// TIA Portal V20 export
TYPE "type_emRelations_em3_sequence"
// stored: Access Published, Namespace Unit1
   STRUCT
      topTapeLoading : Struct
         jobs : "LAF_typeJobs";
         sequence : "LAF_typeSequence";
         selectJobStatus { S7_SetPoint := 'True'} : Array[0..10] of "LAF_typeJobStatus";
         "step" : "LER_typeStep";
         jobInterface : Struct
            chargeJob2 : "LER_typeJobInterface";
         END_STRUCT;
         homeCheck : Struct
            TapeLoadReq { ExternalWritable := 'False'} : Bool;
            TapeLoaded { ExternalWritable := 'False'} : Bool;
         END_STRUCT;
      END_STRUCT;
      topTapeAttachment : Struct
         jobs : "LAF_typeJobs";
         sequence : "LAF_typeSequence";
         selectJobStatus { S7_SetPoint := 'True'} : Array[0..10] of "LAF_typeJobStatus";
         "step" : "LER_typeStep";
         jobInterface : Struct
            tapeGetJob2 : "LER_typeJobInterface";
            tape1PutJob3 : "LER_typeJobInterface";
            tape2PutJob4 : "LER_typeJobInterface";
            tapeIdleJob5 { S7_SetPoint := 'True'} : "LER_typeJobInterface";
         END_STRUCT;
         homeCheck : Struct
            tapeGetReq { ExternalWritable := 'False'} : Bool;
            tapeGet { ExternalWritable := 'False'} : Bool;
         END_STRUCT;
      END_STRUCT;
      topTapeFixStage : Struct
         jobs : "LAF_typeJobs";
         sequence : "LAF_typeSequence";
         selectJobStatus { S7_SetPoint := 'True'} : Array[0..10] of "LAF_typeJobStatus";
         "step" : "LER_typeStep";
         jobInterface : Struct
            loadJob2 : "LER_typeJobInterface";
            taping1Job3 : "LER_typeJobInterface";
            taping2Job4 : "LER_typeJobInterface";
            unloadJob5 : "LER_typeJobInterface";
         END_STRUCT;
         homeCheck : Struct
            partNoDetect { ExternalWritable := 'False'} : Bool;
            partDetect { ExternalWritable := 'False'} : Bool;
         END_STRUCT;
      END_STRUCT;
   END_STRUCT;
   // // topTapeLoading."step".action1[101] : Step[101] : JOB[1] Condition
   // // topTapeLoading."step".action1[110] : Step[110] : Top Tape Loading Backward
   // // topTapeLoading."step".action1[120] : Step[120] : Top Tape Loading Clamp Open
   // // topTapeLoading."step".action1[130] : Step[130] : Top Tape Cutter Up
   // // topTapeLoading."step".action1[140] : Step[140] : Top Tape Cutter Clamp Down
   // // topTapeLoading."step".action1[150] : Step[150] : Top Tape Tension Backward
   // // topTapeLoading."step".action1[190] : Step[190] : JOB[1] Step End
   // // topTapeLoading."step".action1[201] : Step[201] : JOB[2] Condition
   // // topTapeLoading."step".action1[210] : Step[210] : Top Tape Loading Forward & Tension Backward
   // // topTapeLoading."step".action1[220] : Step[220] : Top Tape Clamp Close
   // // topTapeLoading."step".action1[230] : Step[230] : Top Tape Cutter Clamp Up
   // // topTapeLoading."step".action1[240] : Step[240] : Top Tape Loading Backward & Tension Forward
   // // topTapeLoading."step".action1[250] : Step[250] : Top Tape Cutter Clamp Down
   // // topTapeLoading."step".action1[260] : Step[260] : Top Tape Tension Backward
   // // topTapeLoading."step".action1[290] : Step[290] : JOB[2] Step End
   // // topTapeLoading."step".transition1[101] : Step[101] : JOB[1] Condition
   // // topTapeLoading."step".transition1[110] : Step[110] : Top Tape Loading Backward
   // // topTapeLoading."step".transition1[120] : Step[120] : Top Tape Loading Clamp Open
   // // topTapeLoading."step".transition1[130] : Step[130] : Top Tape Cutter Up
   // // topTapeLoading."step".transition1[140] : Step[140] : Top Tape Cutter Clamp Down
   // // topTapeLoading."step".transition1[150] : Step[150] : Top Tape Tension Backward
   // // topTapeLoading."step".transition1[190] : Step[190] : JOB[1] Step End
   // // topTapeLoading."step".transition1[201] : Step[201] : JOB[2] Condition
   // // topTapeLoading."step".transition1[210] : Step[210] : Top Tape Loading Forward & Tension Backward
   // // topTapeLoading."step".transition1[220] : Step[220] : Top Tape Clamp Close
   // // topTapeLoading."step".transition1[230] : Step[230] : Top Tape Cutter Clamp Up
   // // topTapeLoading."step".transition1[240] : Step[240] : Top Tape Loading Backward & Tension Forward
   // // topTapeLoading."step".transition1[250] : Step[250] : Top Tape Cutter Clamp Down
   // // topTapeLoading."step".transition1[260] : Step[260] : Top Tape Tension Backward
   // // topTapeLoading."step".transition1[290] : Step[290] : JOB[2] Step End
   // // topTapeAttachment."step".action1[101] : Step[101] : JOB[1] Condition
   // // topTapeAttachment."step".action1[110] : Step[110] : Attachment Up
   // // topTapeAttachment."step".action1[120] : Step[120] : Top Tape X-Axis Remains Attach Pos
   // // topTapeAttachment."step".action1[130] : Step[130] : Top Tape Attachment Down
   // // topTapeAttachment."step".action1[140] : Step[140] : Top Tape Attachment Vaccum Off
   // // topTapeAttachment."step".action1[150] : Step[150] : Top Tape Attachment Up
   // // topTapeAttachment."step".action1[180] : Step[180] : Top Tape X-Axis Wait Pos
   // // topTapeAttachment."step".action1[190] : Step[190] : JOB[1] Step End
   // // topTapeAttachment."step".action1[201] : Step[201] : JOB[2] Condition
   // // topTapeAttachment."step".action1[210] : Step[210] : Top Tape X-Axis Wait Pos
   // // topTapeAttachment."step".action1[220] : Step[220] : Top Tape Attachment Down
   // // topTapeAttachment."step".action1[230] : Step[230] : Top Tape Attachment Vaccum On
   // // topTapeAttachment."step".action1[240] : Step[240] : Top Tape Cutter Down
   // // topTapeAttachment."step".action1[241] : Step[241] : Top Tape Cutter Up
   // // topTapeAttachment."step".action1[242] : Step[242] : Top Tape Clamp Open
   // // topTapeAttachment."step".action1[250] : Step[250] : Top Tape Attachment Up
   // // topTapeAttachment."step".action1[290] : Step[290] : JOB[2] Step End
   // // topTapeAttachment."step".action1[301] : Step[301] : JOB[3] Condition
   // // topTapeAttachment."step".action1[310] : Step[310] : Top Tape X-Axis Tape-1 Pos
   // // topTapeAttachment."step".action1[320] : Step[320] : Top Tape Attachment Down
   // // topTapeAttachment."step".action1[330] : Step[330] : Top Tape Attachment Vaccum Off
   // // topTapeAttachment."step".action1[370] : Step[370] : Top Tape Attachment Up
   // // topTapeAttachment."step".action1[380] : Step[380] : Top Tape X-Axis Wait Pos
   // // topTapeAttachment."step".action1[390] : Step[390] : JOB[3] Step End
   // // topTapeAttachment."step".action1[401] : Step[401] : JOB[4] Condition
   // // topTapeAttachment."step".action1[410] : Step[410] : Top Tape X-Axis Tape-2 Pos
   // // topTapeAttachment."step".action1[420] : Step[420] : Top Tape Attachment Down
   // // topTapeAttachment."step".action1[430] : Step[430] : Top Tape Attachment Vaccum Off
   // // topTapeAttachment."step".action1[470] : Step[470] : Top Tape Attachment Up
   // // topTapeAttachment."step".action1[480] : Step[480] : Top Tape X-Axis Wait Pos
   // // topTapeAttachment."step".action1[490] : Step[490] : JOB[4] Step End
   // // topTapeAttachment."step".transition1[101] : Step[101] : JOB[1] Condition
   // // topTapeAttachment."step".transition1[110] : Step[110] : Attachment Up
   // // topTapeAttachment."step".transition1[120] : Step[120] : Top Tape X-Axis Remains Attach Pos
   // // topTapeAttachment."step".transition1[130] : Step[130] : Top Tape Attachment Down
   // // topTapeAttachment."step".transition1[140] : Step[140] : Top Tape Attachment Vaccum Off
   // // topTapeAttachment."step".transition1[150] : Step[150] : Top Tape Attachment Up
   // // topTapeAttachment."step".transition1[180] : Step[180] : Top Tape X-Axis Wait Pos
   // // topTapeAttachment."step".transition1[190] : Step[190] : JOB[1] Step End
   // // topTapeAttachment."step".transition1[201] : Step[201] : JOB[2] Condition
   // // topTapeAttachment."step".transition1[210] : Step[210] : Top Tape X-Axis Wait Pos
   // // topTapeAttachment."step".transition1[220] : Step[220] : Top Tape Attachment Down
   // // topTapeAttachment."step".transition1[230] : Step[230] : Top Tape Attachment Vaccum On
   // // topTapeAttachment."step".transition1[240] : Step[240] : Top Tape Cutter Down
   // // topTapeAttachment."step".transition1[241] : Step[241] : Top Tape Cutter Up
   // // topTapeAttachment."step".transition1[242] : Step[242] : Top Tape Clamp Open
   // // topTapeAttachment."step".transition1[250] : Step[250] : Top Tape Attachment Up
   // // topTapeAttachment."step".transition1[290] : Step[290] : JOB[2] Step End
   // // topTapeAttachment."step".transition1[301] : Step[301] : JOB[3] Condition
   // // topTapeAttachment."step".transition1[310] : Step[310] : Top Tape X-Axis Tape-1 Pos
   // // topTapeAttachment."step".transition1[320] : Step[320] : Top Tape Attachment Down
   // // topTapeAttachment."step".transition1[330] : Step[330] : Top Tape Attachment Vaccum Off
   // // topTapeAttachment."step".transition1[370] : Step[370] : Top Tape Attachment Up
   // // topTapeAttachment."step".transition1[380] : Step[380] : Top Tape X-Axis Wait Pos
   // // topTapeAttachment."step".transition1[390] : Step[390] : JOB[3] Step End
   // // topTapeAttachment."step".transition1[401] : Step[401] : JOB[4] Condition
   // // topTapeAttachment."step".transition1[410] : Step[410] : Top Tape X-Axis Tape-2 Pos
   // // topTapeAttachment."step".transition1[420] : Step[420] : Top Tape Attachment Down
   // // topTapeAttachment."step".transition1[430] : Step[430] : Top Tape Attachment Vaccum Off
   // // topTapeAttachment."step".transition1[470] : Step[470] : Top Tape Attachment Up
   // // topTapeAttachment."step".transition1[480] : Step[480] : Top Tape X-Axis Wait Pos
   // // topTapeAttachment."step".transition1[490] : Step[490] : JOB[4] Step End
   // // topTapeFixStage."step".action1[101] : Step[101] : JOB[1] Condition
   // // topTapeFixStage."step".action1[110] : Step[110] : Top Tape Fix Stage Left/Center/Right Top Clamp Up
   // // topTapeFixStage."step".action1[111] : Step[111] : Top Tape Fix Stage Bottom Clamp Down
   // // topTapeFixStage."step".action1[120] : Step[120] : Top Tape Fix Stage Bottom Clamp Up
   // // topTapeFixStage."step".action1[121] : Step[121] : Top Tape Fix Stage Left/Center/Right Top Clamp Down
   // // topTapeFixStage."step".action1[180] : Step[180] : Top Tape Y-Axis Wait Pos
   // // topTapeFixStage."step".action1[190] : Step[190] : JOB[1] Step End
   // // topTapeFixStage."step".action1[201] : Step[201] : JOB[2] Condition
   // // topTapeFixStage."step".action1[210] : Step[210] : Top Tape Fix Stage [Loading Request] => JR PP Left
   // // topTapeFixStage."step".action1[220] : Step[220] Top Tape Y-Axis JR Put/Get Pos
   // // topTapeFixStage."step".action1[230] : Step[230] : Top Tape Fix Stage Bottom Clamp Up
   // // topTapeFixStage."step".action1[231] : Step[231] : Top Tape Fix Stage Left/Center/Right Top Clamp Down
   // // topTapeFixStage."step".action1[232] : Step[232] : Top Tape Fix Stage [Unclamp Request] => JR PP Left
   // // topTapeFixStage."step".action1[270] : Step[270] : Spare
   // // topTapeFixStage."step".action1[280] : Step[280] : Top Tape Y-Axis Wait Pos
   // // topTapeFixStage."step".action1[290] : Step[290] : JOB[2] Step End
   // // topTapeFixStage."step".action1[301] : Step[301] : JOB[3] Conditiion
   // // topTapeFixStage."step".action1[310] : Step[310] : Top Tape Fix Stage => Call Attachment Tape-1
   // // topTapeFixStage."step".action1[320] : Step[320] : Spare
   // // topTapeFixStage."step".action1[390] : Step[390] : JOB[3] Step End
   // // topTapeFixStage."step".action1[401] : Step[401] : JOB[4] Conditiion
   // // topTapeFixStage."step".action1[410] : Step[410] : Top Tape Fix Stage => Call Attachment Tape-1
   // // topTapeFixStage."step".action1[420] : Step[420] : Spare
   // // topTapeFixStage."step".action1[490] : Step[490] : JOB[4] Step End
   // // topTapeFixStage."step".action1[501] : Step[501] : JOB[5] Condition
   // // topTapeFixStage."step".action1[510] : Step[510] : Top Tape Fix Stage [Unloading Request] => JR PP Right
   // // topTapeFixStage."step".action1[520] : Step[520] : Top Tape Fix Stage Y-Axis Put/Get Pos
   // // topTapeFixStage."step".action1[530] : Step[530] : Top Tape Fix Stage [Clamp Request] => JR PP Right
   // // topTapeFixStage."step".action1[531] : Step[531] : Top Tape Fix Stage Left/Center/Right Top Clamp Up
   // // topTapeFixStage."step".action1[532] : Step[532] : Top Tape Fix Stage Bottom Clamp Down
   // // topTapeFixStage."step".action1[570] : Step[570] : Spare
   // // topTapeFixStage."step".action1[580] : Step[580] : Top Tape Y-Axis Wait Pos
   // // topTapeFixStage."step".action1[590] : Step[590] : JOB[5] Step End
   // // topTapeFixStage."step".transition1[101] : Step[101] : JOB[1] Condition
   // // topTapeFixStage."step".transition1[110] : Step[110] : Top Tape Fix Stage Left/Center/Right Top Clamp Up
   // // topTapeFixStage."step".transition1[111] : Step[111] : Top Tape Fix Stage Bottom Clamp Down
   // // topTapeFixStage."step".transition1[120] : Step[120] : Top Tape Fix Stage Bottom Clamp Up
   // // topTapeFixStage."step".transition1[121] : Step[121] : Top Tape Fix Stage Left/Center/Right Top Clamp Down
   // // topTapeFixStage."step".transition1[180] : Step[180] : Top Tape Y-Axis Wait Pos
   // // topTapeFixStage."step".transition1[190] : Step[190] : JOB[1] Step End
   // // topTapeFixStage."step".transition1[201] : Step[201] : JOB[2] Condition
   // // topTapeFixStage."step".transition1[210] : Step[210] : Top Tape Fix Stage [Loading Request] => JR PP Left
   // // topTapeFixStage."step".transition1[220] : Step[220] Top Tape Y-Axis JR Put/Get Pos
   // // topTapeFixStage."step".transition1[230] : Step[230] : Top Tape Fix Stage Bottom Clamp Up
   // // topTapeFixStage."step".transition1[231] : Step[231] : Top Tape Fix Stage Left/Center/Right Top Clamp Down
   // // topTapeFixStage."step".transition1[232] : Step[232] : Top Tape Fix Stage [Unclamp Request] => JR PP Left
   // // topTapeFixStage."step".transition1[270] : Step[270] : Spare
   // // topTapeFixStage."step".transition1[280] : Step[280] : Top Tape Y-Axis Wait Pos
   // // topTapeFixStage."step".transition1[290] : Step[290] : JOB[2] Step End
   // // topTapeFixStage."step".transition1[301] : Step[301] : JOB[3] Conditiion
   // // topTapeFixStage."step".transition1[310] : Step[310] : Top Tape Fix Stage => Call Attachment Tape-1
   // // topTapeFixStage."step".transition1[320] : Step[320] : Spare
   // // topTapeFixStage."step".transition1[390] : Step[390] : JOB[3] Step End
   // // topTapeFixStage."step".transition1[401] : Step[401] : JOB[4] Conditiion
   // // topTapeFixStage."step".transition1[410] : Step[410] : Top Tape Fix Stage => Call Attachment Tape-1
   // // topTapeFixStage."step".transition1[420] : Step[420] : Spare
   // // topTapeFixStage."step".transition1[490] : Step[490] : JOB[4] Step End
   // // topTapeFixStage."step".transition1[501] : Step[501] : JOB[5] Condition
   // // topTapeFixStage."step".transition1[510] : Step[510] : Top Tape Fix Stage [Unloading Request] => JR PP Right
   // // topTapeFixStage."step".transition1[520] : Step[520] : Top Tape Fix Stage Y-Axis Put/Get Pos
   // // topTapeFixStage."step".transition1[530] : Step[530] : Top Tape Fix Stage [Clamp Request] => JR PP Right
   // // topTapeFixStage."step".transition1[531] : Step[531] : Top Tape Fix Stage Left/Center/Right Top Clamp Up
   // // topTapeFixStage."step".transition1[532] : Step[532] : Top Tape Fix Stage Bottom Clamp Down
   // // topTapeFixStage."step".transition1[570] : Step[570] : Spare
   // // topTapeFixStage."step".transition1[580] : Step[580] : Top Tape Y-Axis Wait Pos
   // // topTapeFixStage."step".transition1[590] : Step[590] : JOB[5] Step End
END_TYPE
